SUBAPPLICATION Uebung_020j_AX (* DigitalInput_I1 auf DigitalOutput_Q1/2; 2xAX_TP; Impulsformend *)
  (* Standard: 61499-2; Description: Copyright (c) 2023 Meisterschulen am Ostbahnhof This program and the accompanying materials are made available under the terms of the Eclipse Public License 2.0 which is available at https://www.eclipse.org/legal/epl-2.0/ SPDX-License-Identifier: EPL-2.0 *)
  (* Version 1.0, 2026-01-16, Franz Höpfinger, Meisterschulen am Ostbahnhof, initial API and implementation and/or initial documentation *)
  PACKAGE Uebungen;
  IMPORT logiBUS::io::DI::logiBUS_DI::Input_I1;
  IMPORT logiBUS::io::DQ::logiBUS_DO::Output_Q1;
  IMPORT logiBUS::io::DQ::logiBUS_DO::Output_Q2;
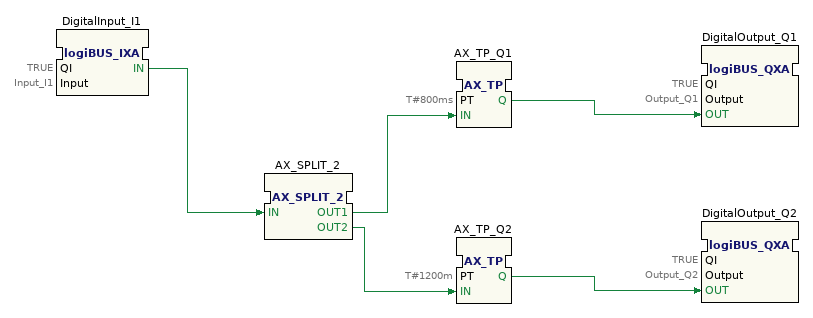
  FBS
    DigitalInput_I1 : logiBUS::io::DI::logiBUS_IXA(QI := TRUE, Input := Input_I1);
    AX_TP_Q1 : adapter::events::unidirectional::timers::AX_TP(PT := T#800ms);
    DigitalOutput_Q1 : logiBUS::io::DQ::logiBUS_QXA(QI := TRUE, Output := Output_Q1);
    AX_TP_Q2 : adapter::events::unidirectional::timers::AX_TP(PT := T#1200m);
    DigitalOutput_Q2 : logiBUS::io::DQ::logiBUS_QXA(QI := TRUE, Output := Output_Q2);
    AX_SPLIT_2 : adapter::events::unidirectional::AX_SPLIT_2;
  END_FBS
  ADAPTER_CONNECTIONS
    AX_TP_Q1.Q TO DigitalOutput_Q1.OUT;
    AX_TP_Q2.Q TO DigitalOutput_Q2.OUT;
    DigitalInput_I1.IN TO AX_SPLIT_2.IN;
    AX_SPLIT_2.OUT1 TO AX_TP_Q1.IN;
    AX_SPLIT_2.OUT2 TO AX_TP_Q2.IN;
  END_CONNECTIONS
END_SUBAPPLICATION
